{attribute 'linkalways'} 
{attribute 'no_explicit_call' := 'This FB is a CLASS and must be accessed using methods or properties'}
{attribute 'enable_dynamic_creation'}
FUNCTION_BLOCK _LINT EXTENDS NumericDatatypeBase
VAR
	localData : LINT;
	activeData : REFERENCE TO LINT REF= localData;
END_VAR

PROPERTY PUBLIC Address : PVOID
GET
Address := ADR(activeData);
END_GET
END_PROPERTY

METHOD PUBLIC ClearReference
VAR_INPUT
END_VAR
activeData REF= localData;
END_METHOD

METHOD PUBLIC Clone : I_Datatype
VAR
    pClone : POINTER TO _LINT;
END_VAR
pClone := __NEW(_LINT(InitialValue := Value));
Clone := pClone^;
END_METHOD

METHOD FB_init : BOOL
VAR_INPUT
	bInitRetains : BOOL; // if TRUE, the retain variables are initialized (warm start / cold start)
	bInCopyCode : BOOL;  // if TRUE, the instance afterwards gets moved into the copy code (online change)
	InitialValue : LINT;
END_VAR
localData := InitialValue;
END_METHOD

PROPERTY PUBLIC IsEven : BOOL
GET
IsEven := (Value mod 2) = 0;
END_GET
END_PROPERTY

PROPERTY PUBLIC IsFloat : BOOL
GET
IsFloat := FALSE;
END_GET
END_PROPERTY

PROPERTY PUBLIC IsSigned : BOOL
GET
IsSigned := TRUE;
END_GET
END_PROPERTY

METHOD PUBLIC MakeReferenceTo
VAR_INPUT
	ReferenceTarget : REFERENCE TO LINT;
END_VAR
activeData REF= ReferenceTarget;
END_METHOD

PROPERTY PUBLIC MaxValue : LINT
GET
MaxValue :=  DatatypeLimits.LINT_MAX_VALUE;
END_GET
END_PROPERTY

PROPERTY PUBLIC MinValue : LINT
GET
MinValue := DatatypeLimits.LINT_MIN_VALUE;
END_GET
END_PROPERTY

METHOD PROTECTED SerializeMaxValue
VAR_INPUT
	Serializer : I_Serializer;
END_VAR
Serializer.AddLint(MaxValue);
END_METHOD

METHOD PROTECTED SerializeMinValue
VAR_INPUT
	Serializer : I_Serializer;
END_VAR
Serializer.AddLint(MinValue);
END_METHOD

METHOD PUBLIC SerializeWith
VAR_INPUT
	Serializer : I_Serializer;
END_VAR
Serializer.AddLint(activeData);
END_METHOD

PROPERTY PUBLIC Size : UDINT
GET
Size := SIZEOF(activeData);
END_GET
END_PROPERTY

METHOD TryDeserializeFrom : BOOL
VAR_INPUT
	Deserializer : I_Deserializer;
	Feedback : I_DeserializerFeedback;
END_VAR
TryDeserializeFrom := Deserializer.TryGetLint(activeData, Feedback);
END_METHOD

METHOD TryMakeReferenceTo : BOOL
VAR_INPUT
	Target : I_Datatype;
END_VAR
VAR
	pTargetData : POINTER TO LINT;
END_VAR
IF NOT (Target.TypeName = TypeName) THEN
	RETURN;
END_IF

pTargetData := Target.Address;
activeData REF= pTargetData^;
TryMakeReferenceTo := TRUE;
END_METHOD

PROPERTY PUBLIC TypeName : T_MAXSTRING
GET
TypeName := 'LINT';
END_GET
END_PROPERTY

PROPERTY PUBLIC Value : REFERENCE TO LINT
GET
Value REF= activeData;
END_GET
END_PROPERTY

END_FUNCTION_BLOCK

(* stored: Version 1.1.0.1, ProductVersion 3.1.4024.13
   POU _LINT: Id {55bb0fd4-1692-4218-9e43-a75a693f6138}, SpecialFunc None
   Folder Constructor: Id {a55fd0c9-47b0-4a24-9ae1-24290dfbf1ba}
   Folder Protected: Id {793ebd05-2562-4524-bdb8-4bfaa81484a1}
   Property Address: Id {0e835d26-7f8a-4302-a460-c82fc62433c9}
   Get Get: Id {3df67f68-1e61-4a39-8308-90e3e5f25fa4}
   Method ClearReference: Id {05c0feaf-a940-4b90-9789-f36dc6191ada}
   Method Clone: Id {ae9d112e-6c70-4015-909f-710417b25570}
   Method FB_init: Id {2d587884-88e9-4ef9-b657-10de24f45edd}
   Property IsEven: Id {f3b4984c-0410-01ff-2951-0361824bfb53}
   Get Get: Id {d66a71b8-3f28-0d92-28b3-f972f6cb713e}
   Property IsFloat: Id {ef4a2020-c2f0-4124-bb89-b212ac73ab4a}
   Get Get: Id {e7b921ea-1173-4677-9b40-e08cf91ba510}
   Property IsSigned: Id {eb322380-9f0c-436e-a490-6777e6a4e06f}
   Get Get: Id {04e57200-a641-446d-921c-4e18d3817201}
   Method MakeReferenceTo: Id {6e230a78-d774-48df-aca2-caa07f3cc9c6}
   Property MaxValue: Id {4689f79f-d282-4b0d-ae12-f82db1c991a3}
   Get Get: Id {b71fa82a-175a-4e27-8ae2-c62f73c29b23}
   Property MinValue: Id {5a4c19d6-4cff-4fb2-a71b-9d936cd51937}
   Get Get: Id {af933da8-ed6e-4a69-b28e-ca9174695f0a}
   Method SerializeMaxValue: Id {fa6b9a02-af1e-42ab-83c1-9e9cf6adc6a5}
   Method SerializeMinValue: Id {72ef36cb-1787-4d44-8996-8f248d8dc992}
   Method SerializeWith: Id {0ef7242e-2aa5-4ce3-94b0-96946b3d223f}
   Property Size: Id {3b83f45d-6d89-4a92-af7e-a15fa24b4842}
   Get Get: Id {8c3e37f0-59bc-48c9-a0e2-d27b70946da9}
   Method TryDeserializeFrom: Id {e839fd22-462e-4ede-bde8-6c9e200e33ea}
   Method TryMakeReferenceTo: Id {00e66337-2827-4cb7-be02-501420604c38}
   Property TypeName: Id {eff9a674-0cff-47b4-a3f7-3835e0803f08}
   Get Get: Id {3b92ecb3-4b18-4433-b975-67d6f02421b8}
   Property Value: Id {87f2d156-b14a-411d-ac91-240bbd247738}
   Get Get: Id {30964aca-f70a-4d8b-9320-ade641e61f61} *)
